Omron Sysmac Studio project TicTacToe2DimensionalArray (Sysmac Studio 1.56.0.64011, StandardProject)

# Controller new_Controller_0: NJ501-1500 version 1.64
Units and slaves: Power Supply : NJ-Px3001; CPU : NJ501-1500
Task PrimaryTask (priority 4, period or condition 1000): Program0

VAR_GLOBAL
    Data_1 : ARRAY[0..2,0..2] OF INT;
    row : INT;
    col : INT;
    Restart : BOOL := False;
    Board : ARRAY[1..3,1..3] OF INT;
    ButtonText : ARRAY[0..3,0..3] of STRING[255];
    Winner : INT;
    WinnerMessage : INT;
    GameStatus : STRING[255];
    CurrentPlayer : INT := 1;
    LineRow1 : BOOL;
    LineRow2 : BOOL;
    LineRow3 : BOOL;
    LineCol1 : BOOL;
    LineCol2 : BOOL;
    LineCol3 : BOOL;
    LineDiag1 : BOOL;
    LineDiag2 : BOOL;
    Button_1 : BOOL;
    Button_2 : BOOL;
    Button_3 : BOOL;
    Button_4 : BOOL;
    Button_5 : BOOL;
    Button_6 : BOOL;
    Button_7 : BOOL;
    Button_8 : BOOL;
    Button_9 : BOOL;
END_VAR

PROGRAM Program0
VAR_EXTERNAL
    Data_1 : ARRAY[0..2,0..2] OF INT;
    row : INT;
    col : INT;
    Restart : BOOL;
    Board : ARRAY[1..3,1..3] OF INT;
    ButtonText : ARRAY[0..3,0..3] of STRING[255];
    Winner : INT;
    WinnerMessage : INT;
    GameStatus : STRING[255];
    CurrentPlayer : INT;
    LineRow1 : BOOL;
    LineRow2 : BOOL;
    LineRow3 : BOOL;
    LineCol1 : BOOL;
    LineCol2 : BOOL;
    LineCol3 : BOOL;
    LineDiag1 : BOOL;
    LineDiag2 : BOOL;
    Button_1 : BOOL;
    Button_2 : BOOL;
    Button_3 : BOOL;
    Button_4 : BOOL;
    Button_5 : BOOL;
    Button_6 : BOOL;
    Button_7 : BOOL;
    Button_8 : BOOL;
    Button_9 : BOOL;
END_VAR

(* Section Section0: ladder, written here as Structured Text *)

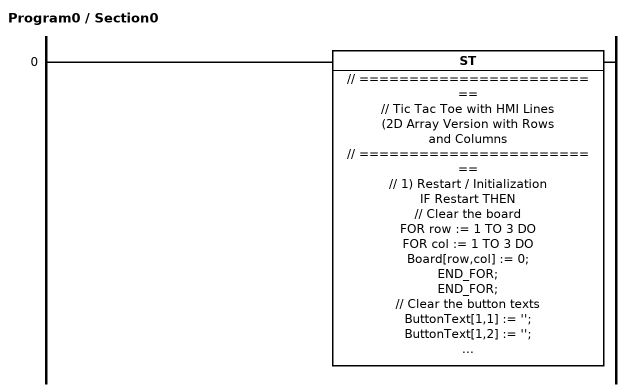
(* Rung 0 *)
// =========================
// Tic Tac Toe with HMI Lines (2D Array Version with Rows and Columns 1-3)
// =========================

// 1) Restart / Initialization
IF Restart THEN
    // Clear the board
    FOR row := 1 TO 3 DO
        FOR col := 1 TO 3 DO
            Board[row,col] := 0;
        END_FOR;
    END_FOR;

    // Clear the button texts
    ButtonText[1,1] := '';
    ButtonText[1,2] := '';
    ButtonText[1,3] := '';
    ButtonText[2,1] := '';
    ButtonText[2,2] := '';
    ButtonText[2,3] := '';
    ButtonText[3,1] := '';
    ButtonText[3,2] := '';
    ButtonText[3,3] := '';

    // Reset game status variables
    Winner := 0;
    WinnerMessage := 0;
    GameStatus := '';
    CurrentPlayer := 1;

    // Reset line indicators
    LineRow1 := FALSE;
    LineRow2 := FALSE;
    LineRow3 := FALSE;
    LineCol1 := FALSE;
    LineCol2 := FALSE;
    LineCol3 := FALSE;
    LineDiag1 := FALSE;
    LineDiag2 := FALSE;

    // Turn off Restart to avoid re-trigger
    Restart := FALSE;
END_IF;

// 2) Allow moves only if no winner yet
IF Winner = 0 THEN
    // Player Move Handling
    IF Button_1 AND (Board[1,1] = 0) THEN
        Board[1,1] := CurrentPlayer;
        IF CurrentPlayer = 1 THEN
            ButtonText[1,1] := 'X';
        ELSE
            ButtonText[1,1] := 'O';
        END_IF;
        CurrentPlayer := 3 - CurrentPlayer;
    END_IF;

    IF Button_2 AND (Board[1,2] = 0) THEN
        Board[1,2] := CurrentPlayer;
        IF CurrentPlayer = 1 THEN
            ButtonText[1,2] := 'X';
        ELSE
            ButtonText[1,2] := 'O';
        END_IF;
        CurrentPlayer := 3 - CurrentPlayer;
    END_IF;

    IF Button_3 AND (Board[1,3] = 0) THEN
        Board[1,3] := CurrentPlayer;
        IF CurrentPlayer = 1 THEN
            ButtonText[1,3] := 'X';
        ELSE
            ButtonText[1,3] := 'O';
        END_IF;
        CurrentPlayer := 3 - CurrentPlayer;
    END_IF;

    IF Button_4 AND (Board[2,1] = 0) THEN
        Board[2,1] := CurrentPlayer;
        IF CurrentPlayer = 1 THEN
            ButtonText[2,1] := 'X';
        ELSE
            ButtonText[2,1] := 'O';
        END_IF;
        CurrentPlayer := 3 - CurrentPlayer;
    END_IF;

    IF Button_5 AND (Board[2,2] = 0) THEN
        Board[2,2] := CurrentPlayer;
        IF CurrentPlayer = 1 THEN
            ButtonText[2,2] := 'X';
        ELSE
            ButtonText[2,2] := 'O';
        END_IF;
        CurrentPlayer := 3 - CurrentPlayer;
    END_IF;

    IF Button_6 AND (Board[2,3] = 0) THEN
        Board[2,3] := CurrentPlayer;
        IF CurrentPlayer = 1 THEN
            ButtonText[2,3] := 'X';
        ELSE
            ButtonText[2,3] := 'O';
        END_IF;
        CurrentPlayer := 3 - CurrentPlayer;
    END_IF;

    IF Button_7 AND (Board[3,1] = 0) THEN
        Board[3,1] := CurrentPlayer;
        IF CurrentPlayer = 1 THEN
            ButtonText[3,1] := 'X';
        ELSE
            ButtonText[3,1] := 'O';
        END_IF;
        CurrentPlayer := 3 - CurrentPlayer;
    END_IF;

    IF Button_8 AND (Board[3,2] = 0) THEN
        Board[3,2] := CurrentPlayer;
        IF CurrentPlayer = 1 THEN
            ButtonText[3,2] := 'X';
        ELSE
            ButtonText[3,2] := 'O';
        END_IF;
        CurrentPlayer := 3 - CurrentPlayer;
    END_IF;

    IF Button_9 AND (Board[3,3] = 0) THEN
        Board[3,3] := CurrentPlayer;
        IF CurrentPlayer = 1 THEN
            ButtonText[3,3] := 'X';
        ELSE
            ButtonText[3,3] := 'O';
        END_IF;
        CurrentPlayer := 3 - CurrentPlayer;
    END_IF;
END_IF;

// 3) Win Detection Logic
// Check rows
IF (Board[1,1] = Board[1,2]) AND (Board[1,2] = Board[1,3]) AND (Board[1,1] <> 0) THEN
    Winner := Board[1,1];
    LineRow1 := TRUE; // Activate line for top row
END_IF;
IF (Board[2,1] = Board[2,2]) AND (Board[2,2] = Board[2,3]) AND (Board[2,1] <> 0) THEN
    Winner := Board[2,1];
    LineRow2 := TRUE; // Middle row
END_IF;
IF (Board[3,1] = Board[3,2]) AND (Board[3,2] = Board[3,3]) AND (Board[3,1] <> 0) THEN
    Winner := Board[3,1];
    LineRow3 := TRUE; // Bottom row
END_IF;

// Check columns
IF (Board[1,1] = Board[2,1]) AND (Board[2,1] = Board[3,1]) AND (Board[1,1] <> 0) THEN
    Winner := Board[1,1];
    LineCol1 := TRUE; // Left column
END_IF;
IF (Board[1,2] = Board[2,2]) AND (Board[2,2] = Board[3,2]) AND (Board[1,2] <> 0) THEN
    Winner := Board[1,2];
    LineCol2 := TRUE; // Middle column
END_IF;
IF (Board[1,3] = Board[2,3]) AND (Board[2,3] = Board[3,3]) AND (Board[1,3] <> 0) THEN
    Winner := Board[1,3];
    LineCol3 := TRUE; // Right column
END_IF;

// Check diagonals
IF (Board[1,1] = Board[2,2]) AND (Board[2,2] = Board[3,3]) AND (Board[1,1] <> 0) THEN
    Winner := Board[1,1];
    LineDiag1 := TRUE; // Main diagonal
END_IF;
IF (Board[1,3] = Board[2,2]) AND (Board[2,2] = Board[3,1]) AND (Board[1,3] <> 0) THEN
    Winner := Board[1,3];
    LineDiag2 := TRUE; // Other diagonal
END_IF;

// 4) Update WinnerMessage & GameStatus
IF Winner = 1 THEN
    WinnerMessage := 1; // Player 1 Wins
    GameStatus := 'Player 1 Wins!';

ELSIF Winner = 2 THEN
    WinnerMessage := 2; // Player 2 Wins
    GameStatus := 'Player 2 Wins!';

ELSIF (Board[1,1] <> 0 AND Board[1,2] <> 0 AND Board[1,3] <> 0 AND
       Board[2,1] <> 0 AND Board[2,2] <> 0 AND Board[2,3] <> 0 AND
       Board[3,1] <> 0 AND Board[3,2] <> 0 AND Board[3,3] <> 0 AND (Winner = 0)) THEN
    WinnerMessage := 0; // It's a Draw
    GameStatus := 'It is a Draw!';
END_IF;
END_PROGRAM

# Device HMI_NA5_0 (NA): not converted